(* IEC 61131-3 sources: RL_MAR/experiments/comparison/llm4plc/results/gpt-4o-mini_20260506_100619/20260506_100907, 3 files *)

(* ---- generated_code_iteration_0.st ---- *)
ructured-text
START_ST
FUNCTION_BLOCK ShellSortFB
VAR_INPUT
    arr: ARRAY[1..1000] OF DINT; // INPUT ARRAY
    sortDirection: BOOL; // SORTING DIRECTION
END_VAR_INPUT

VAR_OUTPUT
    error: BOOL; // ERROR STATUS
    status: WORD; // STATUS CODE
    sorted_arr: ARRAY[1..1000] OF DINT; // OUTPUT SORTED ARRAY
END_VAR_OUTPUT

VAR
    state: INT; // THE STATE VARIABLE
    N: INT := 1000; // ARRAY LENGTH (fixed to 1000)
    i: INT; // LOOP INDEX FOR SHELL SORT
    j: INT; // LOOP INDEX FOR SHELL SORT
    temp: DINT; // TEMPORARY VARIABLE FOR SWAPPING
    gap: INT; // GAP VALUE FOR SHELL SORT
END_VAR

// STATE 0: INITIALIZE
state := 0;
error := FALSE;
status := 16#0000;
FOR i := 1 TO N DO
    sorted_arr[i] := arr[i]; // Copy arr to sorted_arr
END_FOR

// STATE 1: CHECK ARRAY SIZE
IF N <= 1 THEN
    error := TRUE;
    status := 16#8200; // Array size is <= 1
ELSIF N > 1000 THEN
    error := TRUE;
    status := 16#8201; // Array size is > 1000
ELSE
    // STATE 2: SORT ARRAY
    gap := N DIV 2; // Initialize gap
    WHILE gap > 0 DO
        FOR i := gap + 1 TO N DO
            temp := sorted_arr[i];
            j := i;
            WHILE (j > gap) AND ((NOT sortDirection AND sorted_arr[j - gap] > temp) OR (sortDirection AND sorted_arr[j - gap] < temp)) DO
                sorted_arr[j] := sorted_arr[j - gap];
                j := j - gap;
            END_WHILE
            sorted_arr[j] := temp;
        END_FOR
        gap := gap DIV 2; // Reduce gap
    END_WHILE
END_IF

// STATE 3: COMPLETE
state := 3;
END_FUNCTION_BLOCK
END_ST

(* ---- generated_code_iteration_1.st ---- *)
START_REASON
The errors in the original Structured Text (ST) code were primarily due to the incorrect use of variable section terminators. Specifically, the code used "END_VAR_OUTPUT" and "END_VAR_INPUT" to close the variable sections, which is not allowed. Instead, the variable sections should be closed with "END_VAR". This led to the CODESYS compiler validation failure. Additionally, there were no other logical or syntactical errors in the code itself, so the focus will be on correcting the variable section terminators.
END_REASON

START_ST
FUNCTION_BLOCK ShellSortFB
VAR_INPUT
    arr: ARRAY[1..1000] OF DINT; // INPUT ARRAY
    sortDirection: BOOL; // SORTING DIRECTION
END_VAR

VAR_OUTPUT
    error: BOOL; // ERROR STATUS
    status: WORD; // STATUS CODE
    sorted_arr: ARRAY[1..1000] OF DINT; // OUTPUT SORTED ARRAY
END_VAR

VAR
    state: INT; // THE STATE VARIABLE
    N: INT := 1000; // ARRAY LENGTH (fixed to 1000)
    i: INT; // LOOP INDEX FOR SHELL SORT
    j: INT; // LOOP INDEX FOR SHELL SORT
    temp: DINT; // TEMPORARY VARIABLE FOR SWAPPING
    gap: INT; // GAP VALUE FOR SHELL SORT
END_VAR

// STATE 0: INITIALIZE
state := 0;
error := FALSE;
status := 16#0000;
FOR i := 1 TO N DO
    sorted_arr[i] := arr[i]; // Copy arr to sorted_arr
END_FOR

// STATE 1: CHECK ARRAY SIZE
IF N <= 1 THEN
    error := TRUE;
    status := 16#8200; // Array size is <= 1
ELSIF N > 1000 THEN
    error := TRUE;
    status := 16#8201; // Array size is > 1000
ELSE
    // STATE 2: SORT ARRAY
    gap := N DIV 2; // Initialize gap
    WHILE gap > 0 DO
        FOR i := gap + 1 TO N DO
            temp := sorted_arr[i];
            j := i;
            WHILE (j > gap) AND ((NOT sortDirection AND sorted_arr[j - gap] > temp) OR (sortDirection AND sorted_arr[j - gap] < temp)) DO
                sorted_arr[j] := sorted_arr[j - gap];
                j := j - gap;
            END_WHILE
            sorted_arr[j] := temp;
        END_FOR
        gap := gap DIV 2; // Reduce gap
    END_WHILE
END_IF

// STATE 3: COMPLETE
state := 3;
END_FUNCTION_BLOCK
END_ST

(* ---- generated_code_iteration_2.st ---- *)
START_REASON
The errors in the original Structured Text (ST) code were due to the incorrect use of the division operator. The CODESYS compiler requires the use of the semicolon (`;`) instead of the `DIV` operator for integer division in certain contexts. This led to the validation failure. I will replace the `DIV` operator with the appropriate syntax to ensure the code compiles successfully. Additionally, I will ensure that the variable sections are correctly closed with "END_VAR" instead of "END_VAR_OUTPUT" or "END_VAR_INPUT".
END_REASON

START_ST
FUNCTION_BLOCK ShellSortFB
VAR_INPUT
    arr: ARRAY[1..1000] OF DINT; // INPUT ARRAY
    sortDirection: BOOL; // SORTING DIRECTION
END_VAR

VAR_OUTPUT
    error: BOOL; // ERROR STATUS
    status: WORD; // STATUS CODE
    sorted_arr: ARRAY[1..1000] OF DINT; // OUTPUT SORTED ARRAY
END_VAR

VAR
    state: INT; // THE STATE VARIABLE
    N: INT := 1000; // ARRAY LENGTH (fixed to 1000)
    i: INT; // LOOP INDEX FOR SHELL SORT
    j: INT; // LOOP INDEX FOR SHELL SORT
    temp: DINT; // TEMPORARY VARIABLE FOR SWAPPING
    gap: INT; // GAP VALUE FOR SHELL SORT
END_VAR

// STATE 0: INITIALIZE
state := 0;
error := FALSE;
status := 16#0000;
FOR i := 1 TO N DO
    sorted_arr[i] := arr[i]; // Copy arr to sorted_arr
END_FOR

// STATE 1: CHECK ARRAY SIZE
IF N <= 1 THEN
    error := TRUE;
    status := 16#8200; // Array size is <= 1
ELSIF N > 1000 THEN
    error := TRUE;
    status := 16#8201; // Array size is > 1000
ELSE
    // STATE 2: SORT ARRAY
    gap := N / 2; // Initialize gap
    WHILE gap > 0 DO
        FOR i := gap + 1 TO N DO
            temp := sorted_arr[i];
            j := i;
            WHILE (j > gap) AND ((NOT sortDirection AND sorted_arr[j - gap] > temp) OR (sortDirection AND sorted_arr[j - gap] < temp)) DO
                sorted_arr[j] := sorted_arr[j - gap];
                j := j - gap;
            END_WHILE
            sorted_arr[j] := temp;
        END_FOR
        gap := gap / 2; // Reduce gap
    END_WHILE
END_IF

// STATE 3: COMPLETE
state := 3;
END_FUNCTION_BLOCK
END_ST
